PROGRAM MAIN
VAR
	// Lakeshore 224 (Ethernet interface)
	{attribute 'OPC.UA.DA' := '1'}
	LS224_TCP:		FB_LAKESHORE_TCP;		// LakeShore based on FB_TCP_CLIENT
	
	// Lakeshore 336 (Ethernet interface)
	{attribute 'OPC.UA.DA' := '1'}
	LS336_TCP:		FB_LAKESHORE_TCP;		// LakeShore based on FB_TCP_CLIENT


	// Lakeshores to be simulated
	{attribute 'OPC.UA.DA' := '1'}
	LS224_TCP_SIM:		FB_LAKESHORE_TCP;		// LakeShore based on FB_TCP_CLIENT
	{attribute 'OPC.UA.DA' := '1'}
	LS336_TCP_SIM:		FB_LAKESHORE_TCP;		// LakeShore based on FB_TCP_CLIENT

	// Simulators
	SIM_LS224_TCP:	FB_SIM_TCP_LAKESHORE;		// LakeShore SIM based on FB_TCP_SERVER
	SIM_LS336_TCP:	FB_SIM_TCP_LAKESHORE;		// LakeShore SIM based on FB_TCP_SERVER


END_VAR


// Lakeshore 224
LS224_TCP(	in_sName			:= 'LS224_TCP',
			in_nModel			:= 224,
			in_nPeriod			:= 1500,
			in_sCmdSuffix		:= '$0D$0A',
			in_sReplySuffix		:= '$0D$0A',
			in_sDeviceTcpIpAdr	:= '192.168.0.12', 
			in_nDeviceTcpPort	:= 7777);

// Lakeshore 336
LS336_TCP(	in_sName			:= 'LS336_TCP',
			in_nModel			:= 336,
			in_nPeriod			:= 1000,
			in_sCmdSuffix		:= '$0A',
			in_sReplySuffix		:= '$0A',
			in_sDeviceTcpIpAdr	:= '192.168.0.80', 
			in_nDeviceTcpPort	:= 7777);

// Dummy Lakeshore 224
// in_bSimulation:= TRUE means that it communicates with a simulator.
// If the simulator is running on the same PLC, in_sDeviceTcpIpAdr:='127.0.0.1'.
// in_nDeviceTcpPort has to match simulator's in_nTcpPort.
// See SIM_LS224_TCP.
LS224_TCP_SIM(
			in_bSimulation		:= TRUE,	
			in_sName			:= 'LS224_TCP_SIM',
			in_nModel			:= 224,
			in_nPeriod			:= 1500,
			in_sCmdSuffix		:= '$0D$0A',
			in_sReplySuffix		:= '$0D$0A',
			in_sDeviceTcpIpAdr	:= '127.0.0.1', 
			in_nDeviceTcpPort	:= 8888);

// Dummy Lakeshore 336
// in_bSimulation:= TRUE means that it communicates with a simulator.
// If the simulator is running on the same PLC, in_sDeviceTcpIpAdr:='127.0.0.1'.
// in_nDeviceTcpPort has to match simulator's in_nTcpPort.
// See SIM_LS336_TCP.
LS336_TCP_SIM(	
			in_bSimulation		:= TRUE,	
			in_sName			:= 'LS336_TCP_SIM',
			in_nModel			:= 336,
			in_nPeriod			:= 1000,
			in_sCmdSuffix		:= '$0A',
			in_sReplySuffix		:= '$0A',
			in_sDeviceTcpIpAdr	:= '127.0.0.1', 
			in_nDeviceTcpPort	:= 7777);


// Lakeshore simulators
SIM_LS224_TCP(	in_bSimulation	:= TRUE,	
				in_bEnable		:= TRUE, 
				in_nModel		:= 224,
				in_sReplySuffix	:= '$0D$0A',
				in_sTcpIpAdr	:= '127.0.0.1',
				in_nTcpPort		:= 8888);

SIM_LS336_TCP(	in_bSimulation	:= TRUE,	
				in_bEnable		:= TRUE, 
				in_nModel		:= 336, 
				in_sReplySuffix	:= '$0A',
				in_sTcpIpAdr	:= '127.0.0.1',
				in_nTcpPort		:= 7777);

END_PROGRAM

(* stored: Version 1.1.0.1, ProductVersion 3.1.4024.3
   POU MAIN: Id {8a7be1e0-ea1c-46d6-85da-e4fd56afd0df}, SpecialFunc None *)
